FUNCTION_BLOCK FB_Target
VAR_INPUT
END_VAR
VAR_OUTPUT
END_VAR
VAR
END_VAR

END_FUNCTION_BLOCK

(* stored: Version 1.1.0.1, ProductVersion 3.1.4024.12
   POU FB_Target: Id {03a9cd9d-3845-0fb8-3250-b0e6042a4dfc}, SpecialFunc None *)
